# EPICS IOC start-up script: examples/test/PSI/jinja2/loadPLC.iocsh
require ecmccfg,kivel "MASTER_ID=-1"

${SCRIPTEXEC} "${ECMC_CONFIG_ROOT}loadYamlPlc.cmd" "FILE=./plc1.yaml"

# go active
${SCRIPTEXEC} ${ECMC_CONFIG_ROOT}setAppMode.cmd
